// Mitsubishi GX Works2 project: 240927_공급가공분배   PLC: Q03UDV

PROGRAM MAIN
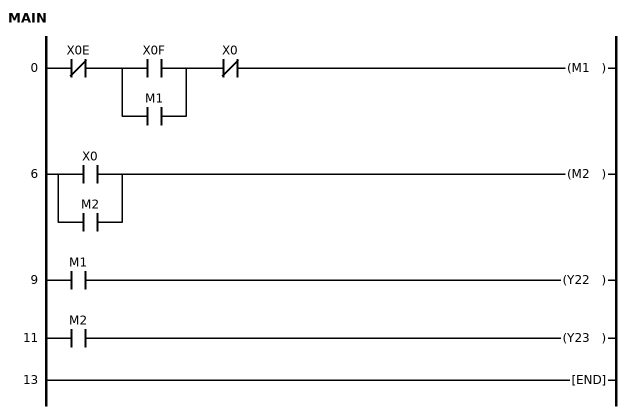
0     LDI     X0E
      LD      X0F
      OR      M1
      ANB
      ANI     X0
      OUT     M1
6     LD      X0
      OR      M2
      OUT     M2
9     LD      M1
      OUT     Y22
11    LD      M2
      OUT     Y23
13    END
END_PROGRAM
